{attribute 'GeneratedUsingTerminal: EL3061-0000-0016'}
{attribute addProperty BoxType "EL3061-0000-0016"}
{attribute addProperty Id "AI_StandardAT %I*AI_Standard_EA9DF21E9WcStateAT %I*WcState_9091E0EB2InfoDataAT %I*InfoData_32EB74EA10"}
{attribute addProperty CRC "1765360954"}
{attribute addProperty Size "21"}
TYPE EL3061_6939453A EXTENDS EtcSlaveTerminalBase_947E5A46 :
STRUCT
	{attribute addProperty Name "AI_Standard"}
	AI_Standard : AI_Standard_EA9DF21E;
	{attribute addProperty Name "WcState"}
	WcState : WcState_9091E0EB;
	{attribute addProperty Name "InfoData"}
	InfoData : InfoData_32EB74EA;
END_STRUCT
END_TYPE

(* stored: Version 1.2.0.0, ProductVersion 3.1.4024.9
   DUT EL3061_6939453A: Id {6000ce84-6c3d-4b41-8e37-f65f3ced37cd} *)
